INTERFACE IFC_ACTUATION

PROPERTY ACCELERATION : LREAL
GET
END_GET
SET
END_SET
END_PROPERTY

METHOD ACTIVATE_EXTERNAL_SETPOINT : DINT
VAR_INPUT
END_VAR
END_METHOD

METHOD ACTIVATE_TOUCHPROBE : DINT
VAR_INPUT
END_VAR
END_METHOD

PROPERTY AT_NEGATIVE_LIMIT : BOOL
GET
END_GET
END_PROPERTY

PROPERTY AT_POSITIVE_LIMIT : BOOL
GET
END_GET
END_PROPERTY

PROPERTY AXIS_ERROR : BOOL
GET
END_GET
END_PROPERTY

PROPERTY AXIS_ERROR_ID : UDINT
GET
END_GET
END_PROPERTY

PROPERTY CALIBRATE_AT_LIMIT : BOOL
GET
END_GET
SET
END_SET
END_PROPERTY

PROPERTY CALIBRATE_TO_NEGATIVE : BOOL
GET
END_GET
SET
END_SET
END_PROPERTY

METHOD DEACTIVATE_EXTERNAL_SETPOINT : DINT
VAR_INPUT
END_VAR
END_METHOD

METHOD DEACTIVATE_TOUCHPROBE : DINT
VAR_INPUT
END_VAR
END_METHOD

PROPERTY DECELERATION : LREAL
GET
END_GET
SET
END_SET
END_PROPERTY

PROPERTY DISABLE_LIMITS : BOOL
GET
END_GET
SET
END_SET
END_PROPERTY

PROPERTY ENABLE : BOOL
GET
END_GET
SET
END_SET
END_PROPERTY

METHOD HALT : DINT
VAR_INPUT
END_VAR
END_METHOD

PROPERTY HARDWARE_ERROR_CODE : UDINT
GET
END_GET
END_PROPERTY

PROPERTY HAS_JOB : BOOL
GET
END_GET
END_PROPERTY

METHOD HOME : DINT
VAR_INPUT
END_VAR
END_METHOD

METHOD HOME_FORCED : DINT
VAR_INPUT
END_VAR
END_METHOD

PROPERTY ID : UDINT
GET
END_GET
END_PROPERTY

PROPERTY INVERT_CALIBRATION_SIGNAL : BOOL
GET
END_GET
SET
END_SET
END_PROPERTY

PROPERTY INVERT_LIMITS : BOOL
GET
END_GET
SET
END_SET
END_PROPERTY

PROPERTY IS_MOVING : BOOL
GET
END_GET
END_PROPERTY

PROPERTY JERK : LREAL
GET
END_GET
SET
END_SET
END_PROPERTY

PROPERTY JOG_BACKWARD : BOOL
SET
END_SET
END_PROPERTY

PROPERTY JOG_FORWARD : BOOL
SET
END_SET
END_PROPERTY

PROPERTY JOG_VELOCITY : LREAL
GET
END_GET
SET
END_SET
END_PROPERTY

PROPERTY MODE : E_ACTUATIONSTATE
GET
END_GET
SET
END_SET
END_PROPERTY

METHOD MOVE_ALONG : LREAL
VAR_INPUT
	VELOCITY	: LREAL;
	FORWARD 	: BOOL;
END_VAR
END_METHOD

METHOD MOVE_BY : DINT
VAR_INPUT
	DISTANCE : LREAL;
	VELOCITY : LREAL;
END_VAR
END_METHOD

METHOD MOVE_TO : DINT
VAR_INPUT
	POSITION : LREAL;
	VELOCITY : LREAL;
END_VAR
END_METHOD

PROPERTY OVERRIDE : LREAL
GET
END_GET
SET
END_SET
END_PROPERTY

PROPERTY POSITION : LREAL
GET
END_GET
END_PROPERTY

METHOD RESET : DINT
VAR_INPUT
END_VAR
END_METHOD

PROPERTY SET_DIRECTION : DINT
SET
END_SET
END_PROPERTY

PROPERTY SET_POSITION : LREAL
SET
END_SET
END_PROPERTY

PROPERTY SET_VELOCITY : LREAL
SET
END_SET
END_PROPERTY

PROPERTY VELOCITY : LREAL
GET
END_GET
END_PROPERTY

END_INTERFACE

(* stored: Version 1.1.0.1, ProductVersion 3.1.4020.3
   Itf IFC_ACTUATION: Id {c02abca6-61fc-4ce6-ab34-832a85e521fb}
   Folder METHODS: Id {9984c8b1-d19f-4d73-8f53-8dfa2a9f2d3c}
   Folder External Set Point: Id {b4fa98c3-d2ad-41b1-92b5-30192acc7147}
   Folder PTP: Id {d9fe3ca2-aaa1-4690-b747-700a1675ec7c}
   Folder Touch Probe: Id {520267be-fadd-4e69-ad3e-f069b620e572}
   Folder PROPERTIES: Id {b01f9d85-f929-4717-9d6a-81a72cd1fe3a}
   Folder Dynamics: Id {96819a23-9e78-4c2c-8025-ef295faeeb47}
   Folder Energise: Id {dd3d4649-d38e-41f5-8c87-02ce8b6563e5}
   Folder Error: Id {e21965f5-b6e1-4cb7-b990-bd78a8ddecbc}
   Folder External Set Point: Id {f58e8ac2-6677-406a-b26a-3ce9c5c61fba}
   Folder Homing: Id {9be0b2c5-a681-4f96-b7e5-3fb7d5446638}
   Folder Info: Id {a0883a98-c39b-4278-8b23-84c65ba2e193}
   Folder Limits: Id {83adca52-c495-49cb-b7ac-2924ab056ff5}
   Folder Manual Movement: Id {f6ee7338-9f5d-4557-bd3f-d7a021b8407d}
   Property ACCELERATION: Id {7062b2d4-780b-4ff2-8313-334af5d46a7f}
   Get Get: Id {e018c663-33be-4183-9816-2c442f775b04}
   Set Set: Id {bf5b2285-ca7b-435a-ab71-e86409ef0415}
   Method ACTIVATE_EXTERNAL_SETPOINT: Id {c2b71442-5ea3-41aa-a8f7-ec75e07c3fed}
   Method ACTIVATE_TOUCHPROBE: Id {94a7c2c8-78c6-4139-82b3-eecf28abee05}
   Property AT_NEGATIVE_LIMIT: Id {03d83d99-0407-431f-a33b-b9f4643cefe9}
   Get Get: Id {6e24a4db-44a2-43d0-8ee8-0f69b3287c35}
   Property AT_POSITIVE_LIMIT: Id {a6dd107a-8b54-4c00-b6db-70fd92e023d3}
   Get Get: Id {a0af2bd2-20fe-4fa5-a655-340b07bbd497}
   Property AXIS_ERROR: Id {051c27f2-35a0-4b42-8663-ff64db66bfa8}
   Get Get: Id {bd7ba178-7f0e-4ca7-95d7-6c0b2abaf056}
   Property AXIS_ERROR_ID: Id {9b0a6bd4-2b10-415e-901b-c517b49349dc}
   Get Get: Id {7ba7ce8e-4e20-4ba1-8861-c625b9042dae}
   Property CALIBRATE_AT_LIMIT: Id {e35182f2-4551-4948-97e3-fb074c03cd2f}
   Get Get: Id {d540a67a-373d-4307-81ce-74db50a44323}
   Set Set: Id {d099080c-94bc-4112-ac61-dde2943051ea}
   Property CALIBRATE_TO_NEGATIVE: Id {336bacc9-9d6d-4902-bb0d-41e24165626a}
   Get Get: Id {d5a8d62c-2e8f-4a3f-be10-ca88119d05b2}
   Set Set: Id {8bb6f7c5-a7b0-4d9e-b4d9-fc2cab65079d}
   Method DEACTIVATE_EXTERNAL_SETPOINT: Id {1ae4155e-5282-4e15-b94b-14b40f1c290b}
   Method DEACTIVATE_TOUCHPROBE: Id {46ac5ff6-874b-4f65-a71c-767ae2685b24}
   Property DECELERATION: Id {0458e6c9-3663-4bdc-9e6c-944d6d29f4ab}
   Get Get: Id {135b7f9c-e49b-4070-913d-0e57fab8109f}
   Set Set: Id {a50b0cd9-ea29-4065-aa40-2668df9371d5}
   Property DISABLE_LIMITS: Id {7977be46-c57d-4b17-894d-8d938fac6199}
   Get Get: Id {885b7fe2-f287-4a11-9b48-aafb3e92f80f}
   Set Set: Id {9f84598c-e5fb-42bd-8770-4e75d3f24ac2}
   Property ENABLE: Id {95706d04-bda9-4954-9299-07e3c53d96fe}
   Get Get: Id {e8e19e4e-27e6-4134-ba3a-5adfe20641b2}
   Set Set: Id {89582159-f599-4c78-ab95-db91c84dfcfa}
   Method HALT: Id {230d3883-ca75-4866-897a-119b810c3b68}
   Property HARDWARE_ERROR_CODE: Id {08633106-e51c-40a3-95cd-54486ead2ec6}
   Get Get: Id {ac49f088-dfdb-4a52-b2f7-ebf6a1411821}
   Property HAS_JOB: Id {1711db1e-9881-42d5-8ecb-1d13d3f78aa7}
   Get Get: Id {cd737e6a-86f1-4ccc-9cd2-d1868a192dc7}
   Method HOME: Id {26e3c30d-a1d8-4765-8ee9-6c408ec274f8}
   Method HOME_FORCED: Id {e4b0e6d3-94f3-4c2d-9886-31d06c9b8457}
   Property ID: Id {1530045a-af52-45bd-a716-68a45c925008}
   Get Get: Id {332afa6a-c103-445c-b330-cc9ef9842e61}
   Property INVERT_CALIBRATION_SIGNAL: Id {e3f71531-938b-45db-8972-f072bfff9c6d}
   Get Get: Id {16940361-5c93-4c90-9f1c-124178279aba}
   Set Set: Id {b179ae3f-3c5d-4d6f-928a-f28b77e08db8}
   Property INVERT_LIMITS: Id {f70f6a59-e41f-4443-8561-ab2c6009ac68}
   Get Get: Id {ae89735c-4435-405e-aed8-d9dab257fda4}
   Set Set: Id {16144c65-8b8b-4fc7-8273-2605df45d57f}
   Property IS_MOVING: Id {46ec3163-e3fd-4552-91ac-b6fb415901ad}
   Get Get: Id {8509c572-39fa-4558-b4b0-e069e08dbb17}
   Property JERK: Id {f499a8ed-10fa-490c-a0d0-d293714ab10f}
   Get Get: Id {e0990dbb-9ebe-48f0-8c29-2be128e5464e}
   Set Set: Id {5dff5a85-eaf2-4f54-b438-8a252d770c73}
   Property JOG_BACKWARD: Id {705bc266-0e01-4cef-bcb4-33f5b1ff7264}
   Set Set: Id {716d8151-2092-47b7-a1d4-0a7b4b4de058}
   Property JOG_FORWARD: Id {2b7fb0c2-cd18-4b0e-9597-52495e3aa920}
   Set Set: Id {b098df23-c23f-485c-81ba-51c034ce0676}
   Property JOG_VELOCITY: Id {2e923b4e-a2f9-40b2-8823-386f3116b9ec}
   Get Get: Id {54ef335c-9481-47fd-922b-bc635172295d}
   Set Set: Id {262380e8-f46a-4353-9c0d-80e7bf3fa98f}
   Property MODE: Id {f6aef5bf-19f5-47d2-a553-6c1b8cca6276}
   Get Get: Id {bebf8923-2bce-4428-abbf-c4908f293a32}
   Set Set: Id {e8c432cb-e7b9-4ada-bde2-6184e9c58331}
   Method MOVE_ALONG: Id {e77cc154-3441-4d7b-8d67-caeca3d9c001}
   Method MOVE_BY: Id {f6de1ac7-e059-412f-815f-6b15438ead8d}
   Method MOVE_TO: Id {9d389a4f-30a9-46ff-ae16-a5d0ce400c1f}
   Property OVERRIDE: Id {e9483a38-6583-4752-b806-6f13961353c0}
   Get Get: Id {7bc50c94-ab76-4d03-9932-56ebc3e42675}
   Set Set: Id {b4f182c4-19e6-42a9-8428-70702fa59e5a}
   Property POSITION: Id {9a1b043e-9e99-474e-83c8-2e030ef3d531}
   Get Get: Id {9f186a46-a4e9-4047-831c-cb8e4695aedd}
   Method RESET: Id {e72d0270-feeb-497d-ad2b-e236201d5e87}
   Property SET_DIRECTION: Id {58524177-2745-447b-97ae-f62f03afe3a1}
   Set Set: Id {c05d40d8-ff08-45dc-a245-62c105c78903}
   Property SET_POSITION: Id {f25db5c6-a5f7-4ef7-a29d-8842f62a83d2}
   Set Set: Id {13127731-c417-4d8e-be3a-d241d96394ad}
   Property SET_VELOCITY: Id {28c6a6b2-ad40-4842-86d5-2e651a3bcd6b}
   Set Set: Id {8bf65ea3-13a6-4b01-8911-ef8a57864f0d}
   Property VELOCITY: Id {e6eccf36-8c9e-44f9-bfdd-7ae00a770400}
   Get Get: Id {719812c2-3b11-4d05-8003-3b5163175030} *)
